// TIA Portal V18 export
FUNCTION "PLC8_910A2_4RTD_IO_Update" : Void   // FC11020, LAD
{ S7_Optimized_Access := 'TRUE' }
VERSION : 0.1
// stored: AutoNumber false, IsIECCheckEnabled false, SetENOAutomatically false, UDAEnableTagReadback false
BEGIN

REGION Network 1: AI1
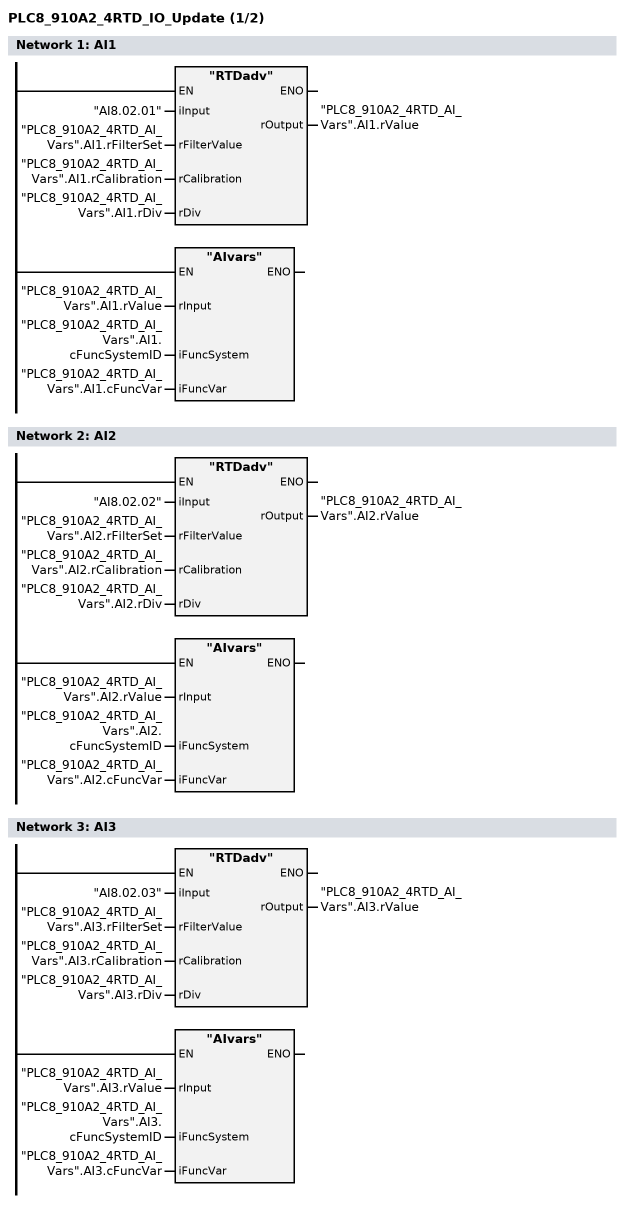
   RUNG wire#powerrail
      "RTDadv"(iInput := "AI8.02.01", rFilterValue := "PLC8_910A2_4RTD_AI_Vars".AI1.rFilterSet, rCalibration := "PLC8_910A2_4RTD_AI_Vars".AI1.rCalibration, rDiv := "PLC8_910A2_4RTD_AI_Vars".AI1.rDiv, rOutput => "PLC8_910A2_4RTD_AI_Vars".AI1.rValue)
   END_RUNG
   RUNG wire#powerrail
      "AIvars"(rInput := "PLC8_910A2_4RTD_AI_Vars".AI1.rValue, iFuncSystem := "PLC8_910A2_4RTD_AI_Vars".AI1.cFuncSystemID, iFuncVar := "PLC8_910A2_4RTD_AI_Vars".AI1.cFuncVar)
   END_RUNG
   // the same network as SCL:
   "RTDadv"(iInput := "AI8.02.01",
            rFilterValue := "PLC8_910A2_4RTD_AI_Vars".AI1.rFilterSet,
            rCalibration := "PLC8_910A2_4RTD_AI_Vars".AI1.rCalibration,
            rDiv := "PLC8_910A2_4RTD_AI_Vars".AI1.rDiv,
            rOutput => "PLC8_910A2_4RTD_AI_Vars".AI1.rValue);
   "AIvars"(rInput := "PLC8_910A2_4RTD_AI_Vars".AI1.rValue,
            iFuncSystem := "PLC8_910A2_4RTD_AI_Vars".AI1.cFuncSystemID,
            iFuncVar := "PLC8_910A2_4RTD_AI_Vars".AI1.cFuncVar);
END_REGION

REGION Network 2: AI2
   RUNG wire#powerrail
      "RTDadv"(iInput := "AI8.02.02", rFilterValue := "PLC8_910A2_4RTD_AI_Vars".AI2.rFilterSet, rCalibration := "PLC8_910A2_4RTD_AI_Vars".AI2.rCalibration, rDiv := "PLC8_910A2_4RTD_AI_Vars".AI2.rDiv, rOutput => "PLC8_910A2_4RTD_AI_Vars".AI2.rValue)
   END_RUNG
   RUNG wire#powerrail
      "AIvars"(rInput := "PLC8_910A2_4RTD_AI_Vars".AI2.rValue, iFuncSystem := "PLC8_910A2_4RTD_AI_Vars".AI2.cFuncSystemID, iFuncVar := "PLC8_910A2_4RTD_AI_Vars".AI2.cFuncVar)
   END_RUNG
   // the same network as SCL:
   "RTDadv"(iInput := "AI8.02.02",
            rFilterValue := "PLC8_910A2_4RTD_AI_Vars".AI2.rFilterSet,
            rCalibration := "PLC8_910A2_4RTD_AI_Vars".AI2.rCalibration,
            rDiv := "PLC8_910A2_4RTD_AI_Vars".AI2.rDiv,
            rOutput => "PLC8_910A2_4RTD_AI_Vars".AI2.rValue);
   "AIvars"(rInput := "PLC8_910A2_4RTD_AI_Vars".AI2.rValue,
            iFuncSystem := "PLC8_910A2_4RTD_AI_Vars".AI2.cFuncSystemID,
            iFuncVar := "PLC8_910A2_4RTD_AI_Vars".AI2.cFuncVar);
END_REGION

REGION Network 3: AI3
   RUNG wire#powerrail
      "RTDadv"(iInput := "AI8.02.03", rFilterValue := "PLC8_910A2_4RTD_AI_Vars".AI3.rFilterSet, rCalibration := "PLC8_910A2_4RTD_AI_Vars".AI3.rCalibration, rDiv := "PLC8_910A2_4RTD_AI_Vars".AI3.rDiv, rOutput => "PLC8_910A2_4RTD_AI_Vars".AI3.rValue)
   END_RUNG
   RUNG wire#powerrail
      "AIvars"(rInput := "PLC8_910A2_4RTD_AI_Vars".AI3.rValue, iFuncSystem := "PLC8_910A2_4RTD_AI_Vars".AI3.cFuncSystemID, iFuncVar := "PLC8_910A2_4RTD_AI_Vars".AI3.cFuncVar)
   END_RUNG
   // the same network as SCL:
   "RTDadv"(iInput := "AI8.02.03",
            rFilterValue := "PLC8_910A2_4RTD_AI_Vars".AI3.rFilterSet,
            rCalibration := "PLC8_910A2_4RTD_AI_Vars".AI3.rCalibration,
            rDiv := "PLC8_910A2_4RTD_AI_Vars".AI3.rDiv,
            rOutput => "PLC8_910A2_4RTD_AI_Vars".AI3.rValue);
   "AIvars"(rInput := "PLC8_910A2_4RTD_AI_Vars".AI3.rValue,
            iFuncSystem := "PLC8_910A2_4RTD_AI_Vars".AI3.cFuncSystemID,
            iFuncVar := "PLC8_910A2_4RTD_AI_Vars".AI3.cFuncVar);
END_REGION

REGION Network 4: AI4
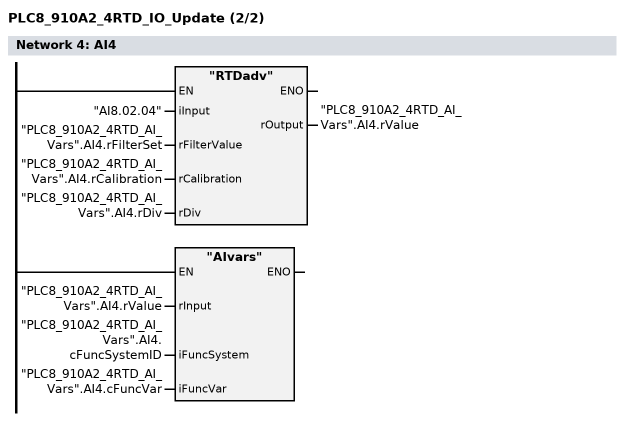
   RUNG wire#powerrail
      "RTDadv"(iInput := "AI8.02.04", rFilterValue := "PLC8_910A2_4RTD_AI_Vars".AI4.rFilterSet, rCalibration := "PLC8_910A2_4RTD_AI_Vars".AI4.rCalibration, rDiv := "PLC8_910A2_4RTD_AI_Vars".AI4.rDiv, rOutput => "PLC8_910A2_4RTD_AI_Vars".AI4.rValue)
   END_RUNG
   RUNG wire#powerrail
      "AIvars"(rInput := "PLC8_910A2_4RTD_AI_Vars".AI4.rValue, iFuncSystem := "PLC8_910A2_4RTD_AI_Vars".AI4.cFuncSystemID, iFuncVar := "PLC8_910A2_4RTD_AI_Vars".AI4.cFuncVar)
   END_RUNG
   // the same network as SCL:
   "RTDadv"(iInput := "AI8.02.04",
            rFilterValue := "PLC8_910A2_4RTD_AI_Vars".AI4.rFilterSet,
            rCalibration := "PLC8_910A2_4RTD_AI_Vars".AI4.rCalibration,
            rDiv := "PLC8_910A2_4RTD_AI_Vars".AI4.rDiv,
            rOutput => "PLC8_910A2_4RTD_AI_Vars".AI4.rValue);
   "AIvars"(rInput := "PLC8_910A2_4RTD_AI_Vars".AI4.rValue,
            iFuncSystem := "PLC8_910A2_4RTD_AI_Vars".AI4.cFuncSystemID,
            iFuncVar := "PLC8_910A2_4RTD_AI_Vars".AI4.cFuncVar);
END_REGION
END_FUNCTION
